{attribute 'GeneratedUsingTerminal: EL1202-0100-0016'}
{attribute addProperty BoxType "EL1202-0100-0016"}
{attribute addProperty Id "NextLatchTimeAT %I*ULINT8"}
{attribute addProperty CRC "443442725"}
{attribute addProperty Size "8"}
TYPE DC_1A6E6625 :
STRUCT
	{attribute addProperty Name "NextLatchTime"}
	NextLatchTime AT %I* : ULINT;
END_STRUCT
END_TYPE

(* stored: Version 1.2.0.0, ProductVersion 3.1.4024.9
   DUT DC_1A6E6625: Id {30789bb4-199b-45c9-ba4b-67c87a72a9a4} *)
